// TwinCAT 3 PLC project Main
// ProgramVersion: 3.1.4023.0
// libraries:
//   Tc2_Standard, * (Beckhoff Automation GmbH)
//   Tc2_System, * (Beckhoff Automation GmbH)
//   Tc2_Utilities, * (Beckhoff Automation GmbH)
//   Tc3_Module, * (Beckhoff Automation GmbH)
//   VisuDialogs, * (System)
//   VisuSymbols,3.5.10.0,System
// project tree:
//   Actuation Systems/Function Blocks/ BulkModulus.TcPOU, DiscreteIntegrator.TcPOU, DiscreteTimeIntegrator_Init.TcPOU, ElectricMotor.TcPOU (not stored), FB_TimeIntegrator.TcPOU (not stored), HPU.TcPOU (not stored), CylinderMech.TcPOU, OrificeEquation.TcPOU, PressureBuildUp.TcPOU (not stored), PressureGradient.TcPOU, Pump.TcPOU (not stored), ValveControlledCylinder.TcPOU, ValveDynamics.TcPOU, VariableBulkModulus.TcPOU (not stored)
//   Actuation Systems/GVL/ FromUnreal.TcGVL (not stored), G_ActuationSystems.TcGVL, Inputs.TcGVL, ToUnreal.TcGVL (not stored), Work.TcGVL
//   Actuation Systems/Programs/ ActuationSystems.TcPOU
//   Functions/ Sign.TcPOU (not stored)
//   / GlobalTextList.TcGTLO, PlcTask.TcTTO, Visualization Manager.TcVMO (not stored)
//   Main Program/ MAIN.TcPOU, P_Joy.TcPOU (not stored)
//   Parameters/ Param.TcGVL, XboxControl.TcGVL (not stored)
//   Parameters/Structs/ Controller.TcDUT (not stored), ST_pValveControlledCylinder.TcDUT
//   VISUs/ Visualization.TcVIS
// real-time tasks:
//   TASK PlcTask: cycle T#1ms, priority 20, ADS port 350

CONFIGURATION Main
    RESOURCE PLC ON TwinCAT3
        TASK PlcTask(INTERVAL := T#1ms, PRIORITY := 20);
        PROGRAM MAIN WITH PlcTask : MAIN;
    END_RESOURCE
END_CONFIGURATION

// ---- Parameters/Structs/ST_pValveControlledCylinder.TcDUT
TYPE ST_pValveControlledCylinder :
STRUCT
	tCycle : LREAL := 1E-4;
	gravity : LREAL := 9.81;	
	Kv : LREAL := 10 / SQRT(7); 						//[L/min / sqrt(bar)]
	DBore : LREAL := 120E-3;							//[m]
	DRod : LREAL := 80E-3;								//[m]
	xMax : LREAL := 1;									//[m]
	x0 : LREAL := 0.5;									//[m]
	pi : LREAL := 3.14159265359;						//Value of pi
    VA0 : LREAL := 0.01;								//[m^3]
	VB0 : LREAL := 0.01;								//[m^3]
	pMax : LREAL := 200E5; 								//[Pa]
	EffectiveMass : LREAL := 5000;						//[kg]
	ExternalForce : LREAL := EffectiveMass*gravity;		//[N]
	FrictionConstant : LREAL := 10000;					//[N/(m/s)]
	pA0 : LREAL := ExternalForce/0.0113;
	pB0 : LREAL := 1E5;
	pAmax : LREAL :=200E5;
	pBmax : LREAL :=200E5;
	vMax : LREAL := 1; 
	v0 : LREAL := 0; 
	OilBulkModulus : LREAL := 12000E5;					//[Pa]
	AdiatricAirConstant : LREAL := 1.4;					//[-]
	AtmosphericPressure : LREAL := 1.01325E5; 			//[Pa]
	VolumetricAirConstant : LREAL := 0.007;				//[%]
	ViscousFrictionCoefficient : LREAL := 1500;			//[kg/s]
	FrictionForceApproximationConstant : LREAL := 250;  //[-]
	ColoumbFriction : LREAL := 75;						//[N] Force
	StaticFrictionForce : LREAL := 500;					//[N]
	StaticFrictionTimeConstant : LREAL := 0.02;			//[s/m]
	cyl_k_end : LREAL := 6E9;                   					//[N/m] spring constant for spring at the stroke limits of a cylinder
	cyl_c_end : LREAL := 9E8;										//[N*s/m] Viscous constant for damper at the stroke limits of a cylinder
END_STRUCT
END_TYPE

// ---- Actuation Systems/GVL/G_ActuationSystems.TcGVL
{attribute 'qualified_only'}
VAR_GLOBAL
ReturnPressure : LREAL;
SupplyPressure : LREAL;
END_VAR

// ---- Actuation Systems/GVL/Inputs.TcGVL
{attribute 'qualified_only'}
VAR_GLOBAL
	uDcvEnableMainJib : BOOL := TRUE;		//Enable/Disable manual control of MainJibCylinder valve
	uDcvMainJib : LREAL;
	uDcvEnableKnuckleJib : BOOL := TRUE;			//Enable/Disable manual control of BoomCylinder valve
	uDcvKnuckleJib : LREAL;
	uDcvEnableKingRotation : BOOL := TRUE;		//Enable/Disable manual control of KingRotationCylinder valve
	uDcvKingRotation : LREAL;
END_VAR

// ---- Actuation Systems/GVL/Work.TcGVL
{attribute 'qualified_only'}
VAR_GLOBAL
	FpistonMainJib : LREAL;
	FpistonKnuckleJib : LREAL;
END_VAR

// ---- Parameters/Param.TcGVL
{attribute 'qualified_only'}
VAR_GLOBAL PERSISTENT
	pMainJibCylinder : ST_pValveControlledCylinder;				//Parameters for MainJibCylinder uses values from ST_pValveControlledCylinder
	pKnuckleJibCylinder : ST_pValveControlledCylinder; 				//Parameters for BoomCylinder uses values from ST_pValveControlledCylinderv
	//pKnuckleCylinder : ST_pValveControlledCylinder;
END_VAR

// ---- Main Program/MAIN.TcPOU
PROGRAM MAIN
VAR
	Timer : LREAL;
END_VAR

//Timer
Timer := Timer + 0.001;

ActuationSystems();
P_Joy();

END_PROGRAM

// ---- Actuation Systems/Programs/ActuationSystems.TcPOU
PROGRAM ActuationSystems
VAR
fbMainJibCylinderHyd : ValveControlledCylinder;
fbKnuckleJibCylinderHyd : ValveControlledCylinder;
fbKingRotationCylinderHyd : ValveControlledCylinder;
//HydraulicCylinder
fbMainJibCylinderMech : CylinderMech;
fbKnuckleJibCylinderMech : CylinderMech;
fbkingRotationCylinderMech : CylinderMech;

fbHPU : HPU;
END_VAR

fbHPU(
);

//Hyd Model for MainJibCylinder
fbMainJibCylinderHyd(
	uDcvEnable := Inputs.uDcvEnableMainJib,
	uDcv := Inputs.uDcvMainJib,	
	ReturnPressure := G_ActuationSystems.ReturnPressure,
	SupplyPressure := G_ActuationSystems.SupplyPressure,
	par := Param.pMainJibCylinder,
	xPiston := FromUnreal.MainJibPistPosition,
	vPiston := FromUnreal.MainJibPistVelocity,
	F_Hydraulic => ToUnreal.MainJibPistForce
);
//Hyd Model for KnuckleJibCylinder
fbKnuckleJibCylinderHyd(
	uDcvEnable := Inputs.uDcvEnableKnuckleJib,
	uDcv := Inputs.uDcvKnuckleJib,	
	ReturnPressure := G_ActuationSystems.ReturnPressure,
	SupplyPressure := G_ActuationSystems.SupplyPressure,
	par := Param.pKnuckleJibCylinder,
	xPiston := fbKnuckleJibCylinderMech.PistonPosition,
	vPiston := fbKnuckleJibCylinderMech.PistonVelocity*1000,
);

//Temp Mechanical Model for MainJibCylinder
fbMainJibCylinderMech(
	F_Hydraulic := fbMainJibCylinderHyd.F_Hydraulic,
	param := Param.pMainJibCylinder,
	F_Piston => Work.FpistonMainJib
);	

fbKnuckleJibCylinderMech(
	F_Hydraulic := fbKnuckleJibCylinderHyd.F_Hydraulic,
	param := Param.pKnuckleJibCylinder,
	F_Piston => Work.FpistonKnuckleJib
);

END_PROGRAM

// ---- Actuation Systems/Function Blocks/ValveControlledCylinder.TcPOU
FUNCTION_BLOCK ValveControlledCylinder
VAR_INPUT
	uDcvEnable : BOOL; 
	uDcv : LREAL;
	ReturnPressure : LREAL;
	SupplyPressure : LREAL;
	par : ST_pValveControlledCylinder;
	xPiston : LREAL;
	vPiston : LREAL;
END_VAR
VAR_OUTPUT
	F_Hydraulic : LREAL;
END_VAR
VAR
	PressurepA : LREAL;
	PressurepB : LREAL;
	
	y_tmp1 : LREAL;
	y_tmp2 : LREAL;
	F_Stribeck_Friction : LREAL;

//Pressure pA
fbPressureGradient_pA : PressureGradient;
//PressurepA : LREAL;

//Pressure pB
fbPressureGradient_pB : PressureGradient;
//PressurepB : LREAL;

//OrificeEquation QA and QB
fbOrificeEquationQ_P_A : OrificeEquation;
fbOrificeEquationQ_B_R : OrificeEquation;
fbOrificeEquationQ_P_B : OrificeEquation;
fbOrificeEquationQ_A_R : OrificeEquation;	
FlowQ_P_A : LREAL;
FlowQ_B_R : LREAL;	
FlowQ_P_B : LREAL;
FlowQ_A_R : LREAL;
FlowQA : LREAL;
FlowQB : LREAL;
FlowQL : LREAL := 0.00001;

//Control
ValveOpeningControl : LREAL := 0.0;
pVelocity : LREAL;

//BulkModulus
fbBulkModulus : BulkModulus;
fbVariableBulkModulus : VariableBulkModulus;

PistonArea : LREAL;
AnnulusArea : LREAL;

//ValveDynamics
fbValveDynamics : ValveDynamics;
uDcvDynamic : LREAL;


END_VAR


//IF uDcvEnable THEN
//	ValveOpeningControl := uDcv;
//ELSE 
//	ValveOpeningControl := 0;
//END_IF

	
PistonArea := EXPT(par.DBore,2) * (par.pi/4.0);
AnnulusArea := (EXPT(par.DBore,2) - EXPT(par.DRod,2)) * (par.pi/4.0);

//ValveOpeningControl := XboxControl.joyLeft;      Commented out xbox control as for now

//ValveDynamics
IF uDcvEnable THEN
	fbValveDynamics(
		udcv_IN := uDcv,
		DynamicValve => ValveOpeningControl
		);
ELSE
	fbValveDynamics(
		udcv_IN := 0,
		DynamicValve => ValveOpeningControl
		);	
END_IF

//VariableBulkModulus
fbVariableBulkModulus(
	OilBulkModulus := par.OilBulkModulus,
	AdiatricAirConstant := par.AdiatricAirConstant,
	AtmosphericPressure := par.AtmosphericPressure,
	VolumetricAirContentOfOil := par.VolumetricAirConstant
	);

//Pressure Gradient pA and Pressure pA
fbPressureGradient_pA(
	TotalVolume := par.VA0 + (xPiston * PistonArea),
	BulkModulus := fbBulkModulus.BulkModulus,
	FlowrateIn := FlowQA,
	FlowrateOut := (vPiston * PistonArea),
	p0 := par.pA0,
	param := par,
	Pressure => PressurepA		
	);

//Pressure Gradient pB and Pressure pB
fbPressureGradient_pB(
	TotalVolume := par.VB0 + ((par.xMax - xPiston) * AnnulusArea),
	BulkModulus := fbBulkModulus.BulkModulus,
	FlowrateIn := (vPiston * AnnulusArea),
	FlowrateOut := FlowQB + FlowQL,
	p0 := par.pB0,
	param := par,
	Pressure => PressurepB		
	);

//Flow through orifices Q_P_A, Q_A_R, Q_B_R, Q_P_B
fbOrificeEquationQ_P_A(
	PressureOut := PressurepA, 			
	PressureIn := SupplyPressure,	
	ValveOpening := ValveOpeningControl,	
	param := par,
	OrificeFlow => FlowQ_P_A
	);
	
fbOrificeEquationQ_A_R(
	PressureOut := ReturnPressure, 			
	PressureIn :=  PressurepA,	
	ValveOpening := ValveOpeningControl,	
	param := par,
	OrificeFlow => FlowQ_A_R
	);

fbOrificeEquationQ_B_R(
	PressureOut := ReturnPressure, 			
	PressureIn := PressurepB,			
	ValveOpening := ValveOpeningControl,
	param := par,
	OrificeFlow => FlowQ_B_R
	);
	
fbOrificeEquationQ_P_B(
	PressureOut := PressurepB, 			
	PressureIn := SupplyPressure,			
	ValveOpening := ValveOpeningControl,
	param := par,
	OrificeFlow => FlowQ_P_B
	);	

IF ValveOpeningControl > 0 THEN
	FlowQA := FlowQ_P_A;		
	FlowQB := FlowQ_B_R;
ELSIF ValveOpeningControl < 0 THEN
	FlowQA := FlowQ_A_R;		
	FlowQB := FlowQ_P_B;
ELSE
	FlowQA := 0.0;		
	FlowQB := 0.0;	
END_IF

// Hydraulic Force [N] //
//// Stribeck Friction Force [N] // Dette går til Urealistisk visualisator
//y_tmp1 := EXP((ABS(vPiston) * par.FrictionForceApproximationConstant) * 2.0);
//y_tmp2 := (y_tmp1 - 1.0) / (y_tmp1 + 1.0);
//F_Stribeck_Friction := (((EXP(( -(vPiston * y_tmp2)) / par.StaticFrictionTimeConstant) * ABS(par.StaticFrictionForce)) + par.ColoumbFriction) * y_tmp2) + (vPiston * par.ViscousFrictionCoefficient);
F_Hydraulic := PressurepA * PistonArea - PressurepB * AnnulusArea;  //F_Stribeck_Friction;
	
//PistonForce Cylinder
//fbPistonForce(
//	PressureBoreSide := PressurepA,
//	PressureRodSide := PressurepB,
//	Aa := PistonArea,
//	Ab := AnnulusArea,
//	PistonPosition := xPiston,
//	PistonVelocity := vPiston,
//	F_Piston => PistonForce
//	);

END_FUNCTION_BLOCK

// ---- Actuation Systems/Function Blocks/PressureGradient.TcPOU
FUNCTION_BLOCK PressureGradient
VAR_INPUT
	TotalVolume: LREAL;
	BulkModulus: LREAL;
	FlowrateIn: LREAL;
	FlowrateOut: LREAL;
	pMax : LREAL;
	p0 : LREAL;
	param : ST_pValveControlledCylinder;
END_VAR
VAR_OUTPUT
	PressureGradient : LREAL;
	Pressure : LREAL;
END_VAR
VAR
	ssMethodType : SINT := 1; 
	fbPressurePascal : DiscreteTimeIntegrator_Init;
END_VAR

 
//PressureGradient in [Pascal/s]
PressureGradient := (FlowrateIn - FlowrateOut) * (BulkModulus / TotalVolume);


//Pressure in [Pascal]
fbPressurePascal(
	ssMethodType := ssMethodType,
	tCycle := param.tCycle,
	In := PressureGradient,
	Init := p0,
	minOut := G_ActuationSystems.ReturnPressure,
	maxOut := param.pAmax,
	Out => Pressure
	);

END_FUNCTION_BLOCK

// ---- Actuation Systems/Function Blocks/BulkModulus.TcPOU
FUNCTION_BLOCK BulkModulus
VAR_INPUT
	OilBulkModulus: LREAL;
	AdiatricAirConstant: LREAL;
	AtmosphericPressure: LREAL;
	CapacitancePressure: LREAL;
	VolumetricAirContentOfOil: LREAL;
END_VAR
VAR_OUTPUT
	BulkModulus : LREAL := 12000E5;
	VariableBulkModulus: LREAL;
END_VAR
VAR
	rtb_Add: LREAL;
END_VAR

rtb_Add := AtmosphericPressure + CapacitancePressure;

VariableBulkModulus := 1.0 / ((1.0 / OilBulkModulus) - (1.0 / ((((VolumetricAirContentOfOil - 1.0) / (EXPT(AtmosphericPressure / rtb_Add, 1.0 / AdiatricAirConstant) * VolumetricAirContentOfOil)) - 1.0) * (rtb_Add * AdiatricAirConstant))));

END_FUNCTION_BLOCK

// ---- Actuation Systems/Function Blocks/DiscreteTimeIntegrator_Init.TcPOU
FUNCTION_BLOCK DiscreteTimeIntegrator_Init
VAR_INPUT
	ssMethodType: SINT;
	In: LREAL;
	Init: LREAL;
	minOut : LREAL;
	maxOut : LREAL;
	tCycle : LREAL;
END_VAR
VAR_OUTPUT
	Out: LREAL;
END_VAR
VAR
	c_DiscreteTimeIntegrator_IC: USINT;
	c_DiscreteTimeIntegrator_DS: LREAL;
END_VAR



CASE ssMethodType OF
    0: 
        (* SystemInitialize for Atomic SubSystem: '<Root>/DiscreteTimeIntegrator_Init' *)
        (* InitializeConditions for DiscreteIntegrator: '<S1>/Discrete-Time Integrator' *)
        c_DiscreteTimeIntegrator_IC := 1;
        (* End of SystemInitialize for SubSystem: '<Root>/DiscreteTimeIntegrator_Init' *)
    1: 
        (* Outputs for Atomic SubSystem: '<Root>/DiscreteTimeIntegrator_Init' *)
        (* DiscreteIntegrator: '<S1>/Discrete-Time Integrator' *)

        IF c_DiscreteTimeIntegrator_IC <> 0 THEN 
            c_DiscreteTimeIntegrator_DS := Init;

            IF c_DiscreteTimeIntegrator_DS >= maxOut THEN 
                c_DiscreteTimeIntegrator_DS := maxOut;
            ELSIF c_DiscreteTimeIntegrator_DS <= minOut THEN 
                c_DiscreteTimeIntegrator_DS := minOut;
            END_IF;

        END_IF;


        IF c_DiscreteTimeIntegrator_DS >= maxOut THEN 
            c_DiscreteTimeIntegrator_DS := maxOut;
        ELSIF c_DiscreteTimeIntegrator_DS <= minOut THEN 
            c_DiscreteTimeIntegrator_DS := minOut;
        END_IF;

       
        Out := c_DiscreteTimeIntegrator_DS;
        
        c_DiscreteTimeIntegrator_IC := 0;
        c_DiscreteTimeIntegrator_DS := (tCycle * In) + c_DiscreteTimeIntegrator_DS;

        IF c_DiscreteTimeIntegrator_DS >= maxOut THEN 
            c_DiscreteTimeIntegrator_DS := maxOut;
        ELSIF c_DiscreteTimeIntegrator_DS <= minOut THEN 
            c_DiscreteTimeIntegrator_DS := minOut;
        END_IF;

END_CASE;

END_FUNCTION_BLOCK

// ---- Actuation Systems/Function Blocks/OrificeEquation.TcPOU
FUNCTION_BLOCK OrificeEquation
VAR_INPUT
	PressureOut: LREAL;
	PressureIn: LREAL;
	ValveOpening: LREAL;
	param : ST_pValveControlledCylinder;
END_VAR
VAR_OUTPUT
	OrificeFlow: LREAL;
END_VAR
VAR
	rtb_Sum: LREAL;
	y: LREAL;
	temp1: LREAL;
	lmin_to_m3s : LREAL;
END_VAR


(* Outputs for Atomic SubSystem: '<Root>/OrificeEquation' *)
(* Sum: '<S1>/Sum' *)
rtb_Sum := (PressureIn - PressureOut)*1E-5;
(* Signum: '<S1>/Sign' *)

IF rtb_Sum < 0.0 THEN 
    y := -1.0;
ELSIF rtb_Sum > 0.0 THEN 
    y := 1.0;
ELSE 
    y := rtb_Sum;
END_IF;

lmin_to_m3s := 1.0/60000.0;

(* End of Signum: '<S1>/Sign' *)

(* Outport: '<Root>/OrificeFlow' incorporates:
 *  Abs: '<S1>/Abs'
 *  Product: '<S1>/Product2'
 *  Sqrt: '<S1>/Sqrt1' *)
temp1 := ABS(rtb_Sum);
OrificeFlow := param.Kv * ValveOpening * y * SQRT(temp1) * lmin_to_m3s;
(* End of Outputs for SubSystem: '<Root>/OrificeEquation' *)

END_FUNCTION_BLOCK

// ---- Actuation Systems/Function Blocks/ValveDynamics.TcPOU
FUNCTION_BLOCK ValveDynamics
VAR_INPUT
	udcv_IN : LREAL;
	wn : LREAL := 30.0;
	dr : LREAL := 0.7;
END_VAR
VAR_OUTPUT
	DynamicValve : LREAL;
END_VAR
VAR
	fDeltaTime : LREAL := 0.001*10;
	fAcceleration : LREAL;
	fbVelocity : FB_TimeIntegrator := (fInit := 0.0);
	fbPosition : FB_TimeIntegrator := (fInit := 0.0);
	a : LREAL;
	b : LREAL;
END_VAR
VAR CONSTANT
END_VAR

//Timer := Timer + 0.001;

////Valve opening signal is sent through this
//DynamicValve := cst1*EXP(-21*Timer)*SIN(cst2*Timer);

IF (wn = 0.0) THEN
	RETURN;
END_IF

a := 1/EXPT(wn, 2.0);
b := dr/wn;

fAcceleration := (udcv_IN - fbVelocity.fOut*b - fbPosition.fOut)/a;

fbVelocity(
	fIn := fAcceleration,
	fStepTime := fDeltaTime,
);

fbPosition(
	fIn := fbVelocity.fOut,
	fStepTime := fDeltaTime,
	bEnableLimits := TRUE,
	fMinVal := -1.0,
	fMaxVal := 1.0,
	fOut => DynamicValve
);

END_FUNCTION_BLOCK

// ---- Actuation Systems/Function Blocks/CylinderMech.TcPOU
FUNCTION_BLOCK CylinderMech
VAR_INPUT
	//PressureBoreSide : LREAL;
	//PressureRodSide : LREAL;
	param : ST_pValveControlledCylinder;
	F_Hydraulic : LREAL;
END_VAR
VAR_OUTPUT
	PistonAcceleration: LREAL;
	PistonVelocity : LREAL;
	PistonPosition : LREAL;
	F_Piston : LREAL;
END_VAR
VAR
	fbPistonVelocity : TimeIntegrator;
	fbPistonPosition : TimeIntegrator;
	fDeltaTime : LREAL := 1E-4;
	y_tmp : LREAL;
	SpringContactCoefficient : LREAL;
	DamperContactCoefficient : LREAL;
	F_Upper_Stroke_Limit : LREAL;
	F_Lower_Stroke_Limit : LREAL;
	F_Stribeck_Friction : LREAL;
	AbsPosition: LREAL;
END_VAR

// Upper Stroke Limit Contact Force [N] //
//IF PistonPosition >= param.xMax THEN 
//	SpringContactCoefficient := param.cyl_k_end;
//ELSIF PistonPosition < param.xMax THEN 
//	SpringContactCoefficient := 0;
//END_IF;	

//IF PistonPosition >= param.xMax THEN 
//	DamperContactCoefficient := param.cyl_c_end;
//ELSIF PistonPosition < param.xMax THEN 
//	DamperContactCoefficient := 0;
//END_IF;	

//F_Upper_Stroke_Limit := ((PistonPosition - param.xMax) * SpringContactCoefficient) + (DamperContactCoefficient * PistonVelocity);



//// Lower Stroke Limit Contact Force [N] //
//IF PistonPosition > 0 THEN 
//	SpringContactCoefficient := 0;
//ELSIF PistonPosition <= 0 THEN 
//	SpringContactCoefficient := param.cyl_k_end;
//END_IF;	

//IF PistonPosition > 0 THEN 
//	DamperContactCoefficient := 0;
//ELSIF PistonPosition <= 0 THEN 
//	DamperContactCoefficient := param.cyl_c_end;
//END_IF;	

//AbsPosition := ABS(PistonPosition);
//F_Lower_Stroke_Limit := (SpringContactCoefficient * AbsPosition) + (DamperContactCoefficient * (-1) * PistonVelocity);



//// Stribeck Friction Force [N] //
y_tmp := EXP((PistonVelocity * param.FrictionForceApproximationConstant) * 2.0);
y_tmp := (y_tmp - 1.0) / (y_tmp + 1.0);
F_Stribeck_Friction := (((EXP(( -(PistonVelocity * y_tmp)) / param.StaticFrictionTimeConstant) * ABS(param.StaticFrictionForce)) + param.ColoumbFriction) * y_tmp) + (PistonVelocity * param.ViscousFrictionCoefficient);


/// Piston Force Total [N] ///
//F_Piston := F_Hydraulic - F_Upper_Stroke_Limit + F_Lower_Stroke_Limit - F_Stribeck_Friction;
F_Piston := F_Hydraulic - F_Stribeck_Friction;


PistonAcceleration := (F_Piston - param.ExternalForce) / param.EffectiveMass;
(* End of Outputs for SubSystem: '<Root>/HydraulicCylinder' *)

fbPistonVelocity(
	fStepTime := fDeltaTime,
	fIn := PistonAcceleration,
	fInit := param.v0,
	fMinVal := -param.vMax,
	fMaxVal := param.vMax,
	fOut => PistonVelocity
	);
	
fbPistonPosition(
	fStepTime := param.tCycle,
	fIn := PistonVelocity,
	fInit := param.x0,
	fMinVal := 0,
	fMaxVal := param.xMax,
	fOut => PistonPosition
	);

	//The 2 below uses the old DiscreteTimeIntegrator_Init FB
//fbPistonVelocity(
//	ssMethodType := ssMethodType,
//	tCycle := param.tCycle,
//	In := PistonAcceleration,
//	Init := param.v0,
//	minOut := -param.vMax,
//	maxOut := param.vMax,
//	Out => PistonVelocity
//	);
	
//fbPistonPosition(
//	ssMethodType := ssMethodType,
//	tCycle := param.tCycle,
//	In := PistonVelocity,
//	Init := param.x0,
//	minOut := 0,
//	maxOut := param.xMax,
//	Out => PistonPosition
//	);

//IF PistonPosition >= param.xMax THEN 
//	PistonPosition := param.xMax;
//ELSIF PistonPosition <= 0 THEN 
//	PistonPosition := 0;
//END_IF;

END_FUNCTION_BLOCK

// ---- Actuation Systems/Function Blocks/DiscreteIntegrator.TcPOU
FUNCTION_BLOCK DiscreteIntegrator
VAR_INPUT
	ssMethodType: SINT;
	In1: LREAL;
	StepTime : LREAL := 0.001*10;
END_VAR
VAR_OUTPUT
	Out1: LREAL;
END_VAR
VAR
	c_DiscreteIntegratorMain_DS: LREAL;
	k1: LREAL := 1.0;

END_VAR



CASE ssMethodType OF
    0: 
        (* SystemInitialize for Atomic SubSystem: '<Root>/DiscreteIntegrator' *)
        (* InitializeConditions for DiscreteIntegrator: '<S1>/DiscreteIntegratorMain' *)
        c_DiscreteIntegratorMain_DS := 0.0;
        (* End of SystemInitialize for SubSystem: '<Root>/DiscreteIntegrator' *)
    1: 
        (* Outputs for Atomic SubSystem: '<Root>/DiscreteIntegrator' *)
        (* Outport: '<Root>/Out1' incorporates:
         *  DiscreteIntegrator: '<S1>/DiscreteIntegratorMain' *)
        Out1 := c_DiscreteIntegratorMain_DS;
        (* Update for DiscreteIntegrator: '<S1>/DiscreteIntegratorMain' incorporates:
         *  Gain: '<S1>/Gain' *)
        c_DiscreteIntegratorMain_DS := ((k1 * In1) * StepTime) + c_DiscreteIntegratorMain_DS;
        (* End of Outputs for SubSystem: '<Root>/DiscreteIntegrator' *)
		

END_CASE;

END_FUNCTION_BLOCK

// ---- GlobalTextList.TcGTLO
TEXTLIST GlobalTextList
  353 = '\t\t'
  398 = '%0.1f'
  566 = '%0.2f'
  627 = '%0.5f'
  37 = '%1f'
  729 = '%2f'
  210 = '%f'
  342 = '%f [-]'
  839 = '%f.2'
  735 = '%f0.2'
  760 = '%f0.5'
  189 = '%f2'
  842 = '0'
  160 = 'King Cylinder Rotation'
  808 = 'King Cylinder Rotation\n< -1,1 > '
  413 = 'KingRotation Cylinder Position\n< -1,1 > '
  270 = 'KingRotation Valve Controls'
  72 = 'KnuckleBoom Cylinder Position'
  993 = 'KnuckleBoom Cylinder Position\n< -1,1 > '
  875 = 'KnuckleBoom Valve Controls'
  610 = 'MainBoom Cylinder Position'
  758 = 'MainBoom Cylinder Position\n< -1,1 > '
  351 = 'MainBoom Cylinder Position\nd'
  844 = 'MainBoom Cylinder Position '
  334 = 'MainBoom Cylinder Position                                             Min 2'
  503 = 'MainBoom Valve Controls'
  434 = 'MainBoomCylinderOpe'
  81 = 'uDCV'
  164 = 'uDCV:'
  387 = 'Valve Control Enable'
  112 = 'Valve Control Enable/Reset'
  159 = 'Valve Control Enable:'
  716 = 'x = 0'
END_TEXTLIST

// ---- VISUs/Visualization.TcVIS
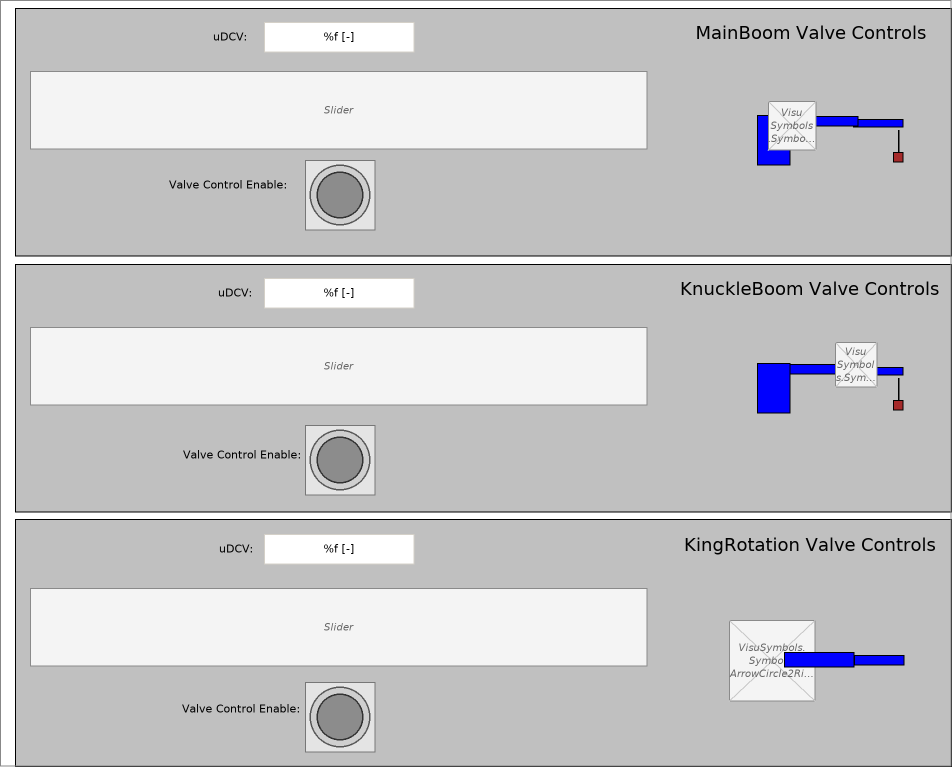
VISUALIZATION Visualization  // 952x767
    RoundedRectangle (15,519 937x248)
    RoundedRectangle (15,264 937x248)
    RoundedRectangle (15,8 937x248)
    Slider (30,71 617x78), variable: Inputs.uDcvMainJib, scale -1..1
    PushSwitchLed (305,160 70x70), variable: Inputs.uDcvEnableMainJib, behaviour: TOGGLE, style: Switch-PushSwitchLed-Gray
    Textfield (264,22 150x30), "%f [-]", text variable: Inputs.uDcvMainJib
        OnMouseClick: write the text variable via Default, min -1, max 1
    Label (197,22 66x30), "uDCV:"
    Label (137,170 182x30), "Valve Control Enable:"
    Slider (30,327 617x78), variable: Inputs.uDcvKnuckleJib, scale -1..1
    PushSwitchLed (305,425 70x70), variable: Inputs.uDcvEnableKnuckleJib, behaviour: TOGGLE, style: Switch-PushSwitchLed-Gray
    Textfield (264,278 150x30), "%f [-]", text variable: Inputs.uDcvKnuckleJib
        OnMouseClick: write the text variable via Default, min -1, max 1
    Label (202,278 66x30), "uDCV:"
    Label (151,440 182x30), "Valve Control Enable:"
    Label (676,18 270x30), "MainBoom Valve Controls"
    Label (675,274 270x30), "KnuckleBoom Valve Controls"
    Slider (30,588 617x78), variable: Inputs.uDcvKingRotation, scale -1..1
    PushSwitchLed (305,682 70x70), variable: Inputs.uDcvEnableKingRotation, behaviour: TOGGLE, style: Switch-PushSwitchLed-Gray
    Textfield (264,534 150x30), "%f [-]", text variable: Inputs.uDcvKingRotation
        OnMouseClick: write the text variable via Default, min -1, max 1
    Label (203,534 66x30), "uDCV:"
    Label (150,694 182x30), "Valve Control Enable:"
    Label (675,530 270x30), "KingRotation Valve Controls"
    Ellipse (757,645 30x30)
    Image (729,620 86x81), angle 320, image: VisuSymbols.Symbols.ArrowCircle2RightRightLeft
    Rectangle (854,655 50x10)
    Rectangle (784,652 70x15)
    Rectangle (887,389 22x1), angle 270
    Rectangle (853,367 50x8), angle 203
    Rectangle (788,364 70x10), angle 349
    Rectangle (757,363 33x50)
    Rectangle (893,400 10x10)
    Rectangle (757,115 33x50)
    Rectangle (887,141 22x1), angle 270
    Rectangle (853,119 50x8), angle 203
    Rectangle (788,116 70x10), angle 349
    Rectangle (893,152 10x10)
    Image (768,101 48x49), angle 345, image: VisuSymbols.Symbols.ArrowCircle2LeftUpDown
    Image (835,342 42x45), angle 10, image: VisuSymbols.Symbols.ArrowCircle2LeftUpDown
END_VISUALIZATION
